// TIA Portal V19 export
TYPE "StatusArea"
// stored: Access Published
   STRUCT
      WarningPresence : Bool;   // Cumulative warning presence
      AlarmPresence : Bool;   // Cumulative alarm presence
      WarningsNumber : Int;   // Active alarms number
      AlarmsNumber : Int;   // Active warnings number
      Status : Int;   // Status from area
   END_STRUCT;
END_TYPE
